// SIMATIC S7-200 project (STEP 7-Micro/WIN), CPU 221 REL 01.10

SYMBOL_TABLE 用户定义1
启动               I0.0
下限开关             I0.1
上限开关             I0.2
右限开关             I0.3
左限开关             I0.4
下降指示             Q0.0
夹紧指示             Q0.1
上升指示             Q0.2
右移指示             Q0.3
左移指示             Q0.4
原位指示             Q0.5
END_SYMBOL_TABLE

ORGANIZATION_BLOCK 主程序:OB1
TITLE=程序注释
BEGIN
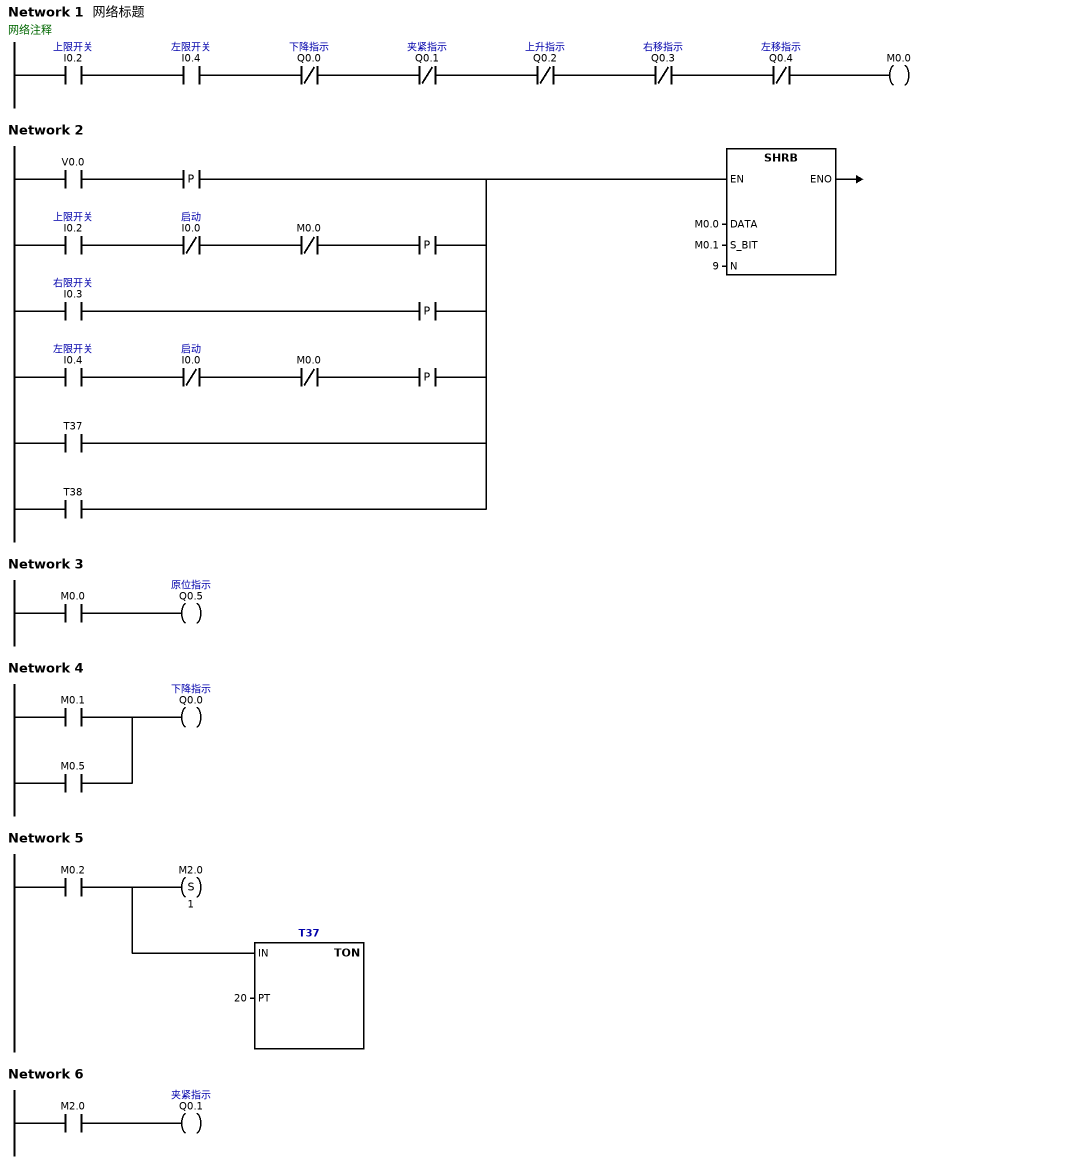
Network 1 // 网络标题
// 网络注释
LD     上限开关:I0.2
A      左限开关:I0.4
AN     下降指示:Q0.0
AN     夹紧指示:Q0.1
AN     上升指示:Q0.2
AN     右移指示:Q0.3
AN     左移指示:Q0.4
=      M0.0
Network 2
// (network saved uncompiled; LAD cells follow)
// row 0: c0 -| |- V0.0  c1 -|P|-  c2 --  c3 -- v  c4 --  c5 --  c6 [SHRB EN:=power@row0, DATA:=M0.0, S_BIT:=M0.1, N:=9, ENO=>power]  c7 ->
// row 1: c0 -| |- 上限开关:I0.2  c1 -|/|- 启动:I0.0  c2 -|/|- M0.0  c3 -|P|-  ^v  c6 [box]
// row 2: c0 -| |- 右限开关:I0.3  c1 --  c2 --  c3 -|P|-  ^v
// row 3: c0 -| |- 左限开关:I0.4  c1 -|/|- 启动:I0.0  c2 -|/|- M0.0  c3 -|P|-  ^v
// row 4: c0 -| |- T37  c1 --  c2 --  c3 -- ^v
// row 5: c0 -| |- T38  c1 --  c2 --  c3 -- ^
Network 3
LD     M0.0
=      原位指示:Q0.5
Network 4
LD     M0.1
O      M0.5
=      下降指示:Q0.0
Network 5
LD     M0.2
S      M2.0, 1
TON    T37, 20
Network 6
LD     M2.0
=      夹紧指示:Q0.1
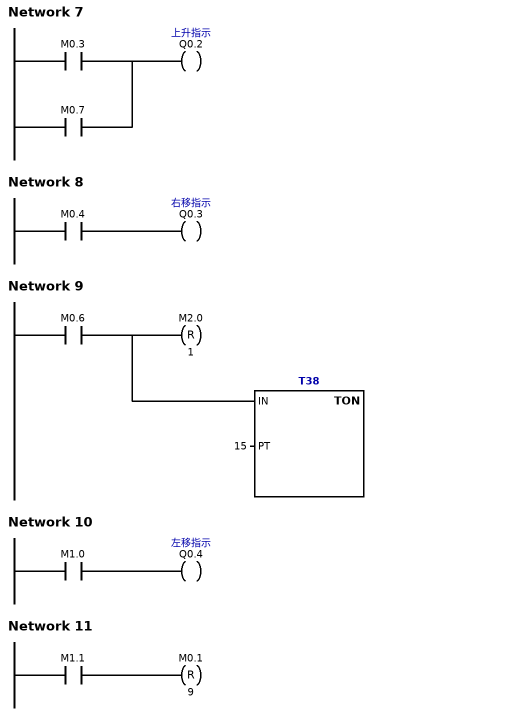
Network 7
LD     M0.3
O      M0.7
=      上升指示:Q0.2
Network 8
LD     M0.4
=      右移指示:Q0.3
Network 9
LD     M0.6
R      M2.0, 1
TON    T38, 15
Network 10
LD     M1.0
=      左移指示:Q0.4
Network 11
LD     M1.1
R      M0.1, 9
END_ORGANIZATION_BLOCK
